TYPE St_Event :
STRUCT
	eEventType : E_EventType;
	eVentSeverity : TcEventSeverity;
	nEventIdentity : UDINT;
	SEventText : STRING(255);
	dtTimeStamp : DATE_AND_TIME;
END_STRUCT
END_TYPE

(* stored: Version 1.1.0.1, ProductVersion 3.1.4024.12
   DUT St_Event: Id {de560a14-9aa9-466e-8324-17ea4a4fba17} *)
